Staubli VAL3: powerOff.pgx

program powerOff()
begin
  disablePower()
  message="disablePower:done"
  taskCreate "sendStatus",100,sendStatus()
  taskKill ("powerOff")
end
